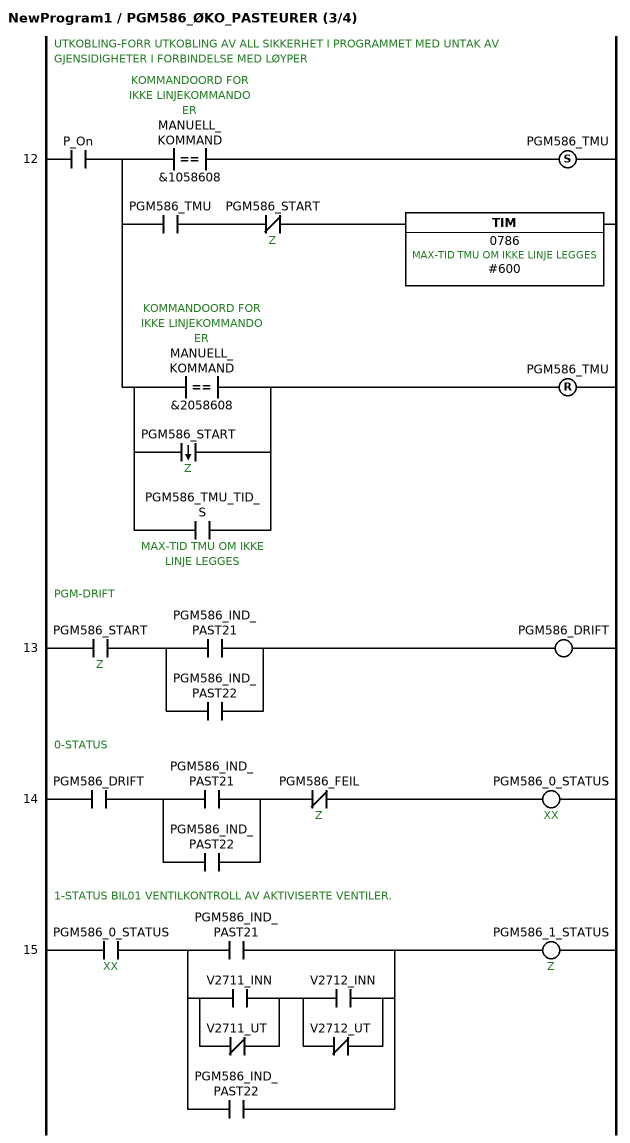
; [picture p720: NewProgram1 / PGM586_ØKO_PASTEURER, rungs 12-15]
; rung 12: UTKOBLING-FORR UTKOBLING AV ALL SIKKERHET I PROGRAMMET MED UNTAK AV GJENSIDIGHETER I FORBINDELSE MED LØYPER
LD P_On
OUT TR0
AND=L(301) MANUELL_KOMMAND &1058608  ; KOMMANDOORD FOR IKKE LINJEKOMMANDOER
SET PGM586_TMU
LD TR0
AND PGM586_TMU
ANDNOT PGM586_START  ; Z
TIM 0786 #600  ; MAX-TID TMU OM IKKE LINJE LEGGES
LD TR0
LD=L(301) MANUELL_KOMMAND &2058608  ; KOMMANDOORD FOR IKKE LINJEKOMMANDOER
%OR PGM586_START  ; Z
OR PGM586_TMU_TID_S  ; MAX-TID TMU OM IKKE LINJE LEGGES
ANDLD
RSET PGM586_TMU
; rung 13: PGM-DRIFT
LD PGM586_START  ; Z
LD PGM586_IND_PAST21
OR PGM586_IND_PAST22
ANDLD
OUT PGM586_DRIFT
; rung 14: 0-STATUS
LD PGM586_DRIFT
LD PGM586_IND_PAST21
OR PGM586_IND_PAST22
ANDLD
ANDNOT PGM586_FEIL  ; Z
OUT PGM586_0_STATUS  ; XX
; rung 15: 1-STATUS BIL01 VENTILKONTROLL AV AKTIVISERTE VENTILER.
LD PGM586_0_STATUS  ; XX
LD PGM586_IND_PAST21
LD V2711_INN
ORNOT V2711_UT
LD V2712_INN
ORNOT V2712_UT
ANDLD
ORLD
OR PGM586_IND_PAST22
ANDLD
OUT PGM586_1_STATUS  ; Z

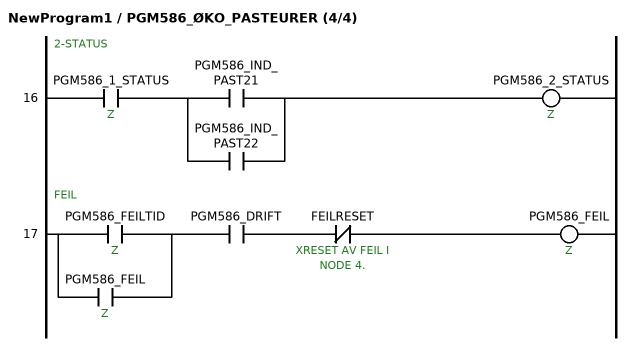
; rung 16: 2-STATUS
LD PGM586_1_STATUS  ; Z
LD PGM586_IND_PAST21
OR PGM586_IND_PAST22
ANDLD
OUT PGM586_2_STATUS  ; Z
; rung 17: FEIL
LD PGM586_FEILTID  ; Z
OR PGM586_FEIL  ; Z
AND PGM586_DRIFT
ANDNOT FEILRESET  ; XRESET AV FEIL I NODE 4.
OUT PGM586_FEIL  ; Z
; rung 18: Ingen_kommentar_funnet

### Section PGM587_RÅMELKSDRENERING

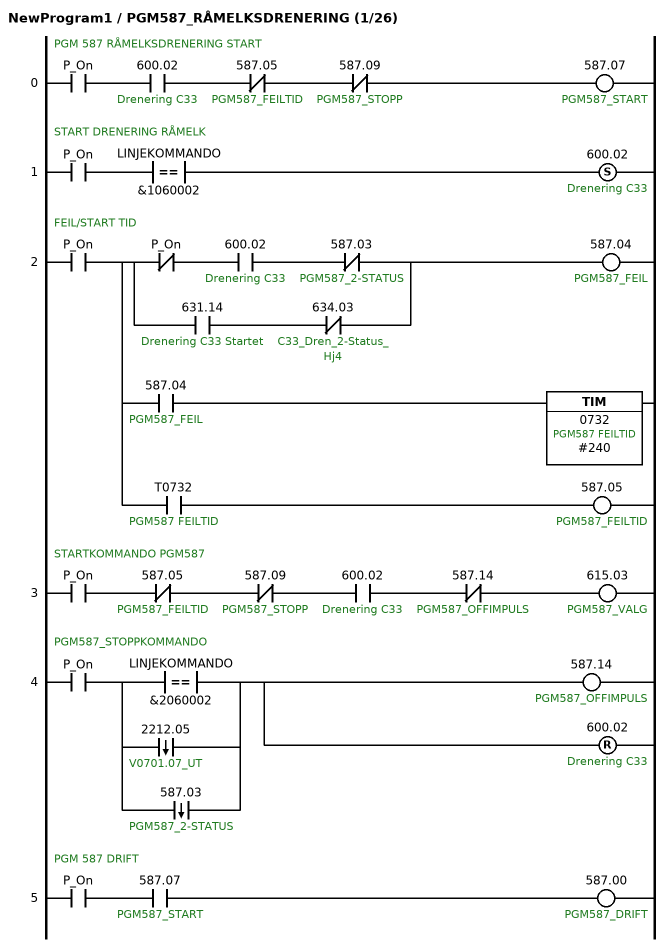
; rung 0: PGM 587 RÅMELKSDRENERING START
LD P_On
AND 600.02  ; Drenering C33
ANDNOT 587.05  ; PGM587_FEILTID
ANDNOT 587.09  ; PGM587_STOPP
OUT 587.07  ; PGM587_START
; rung 1: START DRENERING RÅMELK
LD P_On
AND=L(301) LINJEKOMMANDO &1060002
SET 600.02  ; Drenering C33
; rung 2: FEIL/START TID
LD P_On
OUT TR0
LDNOT P_On
AND 600.02  ; Drenering C33
ANDNOT 587.03  ; PGM587_2-STATUS
LD 631.14  ; Drenering C33 Startet
ANDNOT 634.03  ; C33_Dren_2-Status_Hj4
ORLD
ANDLD
OUT 587.04  ; PGM587_FEIL
LD TR0
AND 587.04  ; PGM587_FEIL
TIM 0732 #240  ; PGM587 FEILTID
LD TR0
AND T0732  ; PGM587 FEILTID
OUT 587.05  ; PGM587_FEILTID
; rung 3: STARTKOMMANDO PGM587
LD P_On
ANDNOT 587.05  ; PGM587_FEILTID
ANDNOT 587.09  ; PGM587_STOPP
AND 600.02  ; Drenering C33
ANDNOT 587.14  ; PGM587_OFFIMPULS
OUT 615.03  ; PGM587_VALG
; rung 4: PGM587_STOPPKOMMANDO
LD P_On
LD=L(301) LINJEKOMMANDO &2060002
%OR 2212.05  ; V0701.07_UT
%OR 587.03  ; PGM587_2-STATUS
ANDLD
OUT 587.14  ; PGM587_OFFIMPULS
RSET 600.02  ; Drenering C33
; rung 5: PGM 587 DRIFT
LD P_On
AND 587.07  ; PGM587_START
OUT 587.00  ; PGM587_DRIFT

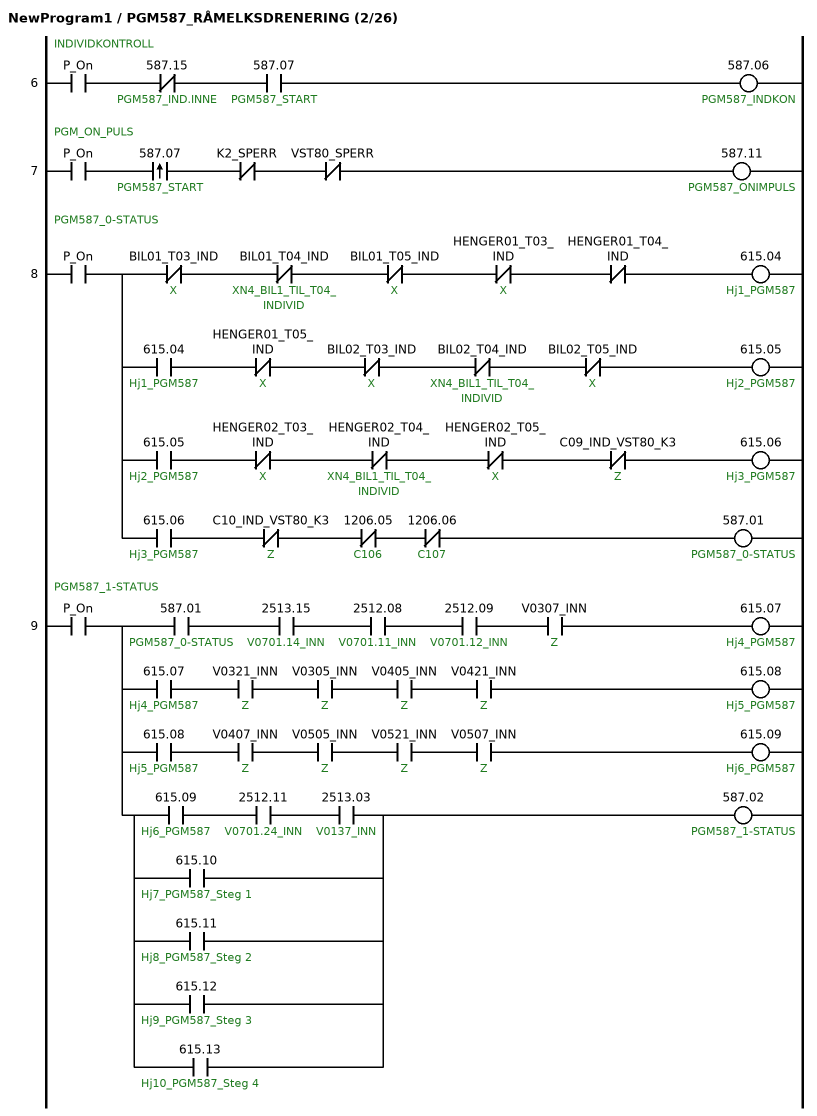
; rung 6: INDIVIDKONTROLL
LD P_On
ANDNOT 587.15  ; PGM587_IND.INNE
AND 587.07  ; PGM587_START
OUT 587.06  ; PGM587_INDKON
; rung 7: PGM_ON_PULS
LD P_On
@AND 587.07  ; PGM587_START
ANDNOT K2_SPERR
ANDNOT VST80_SPERR
OUT 587.11  ; PGM587_ONIMPULS
; rung 8: PGM587_0-STATUS
LD P_On
OUT TR0
ANDNOT BIL01_T03_IND  ; X
ANDNOT BIL01_T04_IND  ; XN4_BIL1_TIL_T04_INDIVID
ANDNOT BIL01_T05_IND  ; X
ANDNOT HENGER01_T03_IND  ; X
ANDNOT HENGER01_T04_IND
OUT 615.04  ; Hj1_PGM587
LD TR0
AND 615.04  ; Hj1_PGM587
ANDNOT HENGER01_T05_IND  ; X
ANDNOT BIL02_T03_IND  ; X
ANDNOT BIL02_T04_IND  ; XN4_BIL1_TIL_T04_INDIVID
ANDNOT BIL02_T05_IND  ; X
OUT 615.05  ; Hj2_PGM587
LD TR0
AND 615.05  ; Hj2_PGM587
ANDNOT HENGER02_T03_IND  ; X
ANDNOT HENGER02_T04_IND  ; XN4_BIL1_TIL_T04_INDIVID
ANDNOT HENGER02_T05_IND  ; X
ANDNOT C09_IND_VST80_K3  ; Z
OUT 615.06  ; Hj3_PGM587
LD TR0
AND 615.06  ; Hj3_PGM587
ANDNOT C10_IND_VST80_K3  ; Z
ANDNOT 1206.05  ; C106
ANDNOT 1206.06  ; C107
OUT 587.01  ; PGM587_0-STATUS
; rung 9: PGM587_1-STATUS
LD P_On
OUT TR0
AND 587.01  ; PGM587_0-STATUS
AND 2513.15  ; V0701.14_INN
AND 2512.08  ; V0701.11_INN
AND 2512.09  ; V0701.12_INN
AND V0307_INN  ; Z
OUT 615.07  ; Hj4_PGM587
LD TR0
AND 615.07  ; Hj4_PGM587
AND V0321_INN  ; Z
AND V0305_INN  ; Z
AND V0405_INN  ; Z
AND V0421_INN  ; Z
OUT 615.08  ; Hj5_PGM587
LD TR0
AND 615.08  ; Hj5_PGM587
AND V0407_INN  ; Z
AND V0505_INN  ; Z
AND V0521_INN  ; Z
AND V0507_INN  ; Z
OUT 615.09  ; Hj6_PGM587
LD TR0
LD 615.09  ; Hj6_PGM587
AND 2512.11  ; V0701.24_INN
AND 2513.03  ; V0137_INN
OR 615.10  ; Hj7_PGM587_Steg 1
OR 615.11  ; Hj8_PGM587_Steg 2
OR 615.12  ; Hj9_PGM587_Steg 3
OR 615.13  ; Hj10_PGM587_Steg 4
ANDLD
OUT 587.02  ; PGM587_1-STATUS

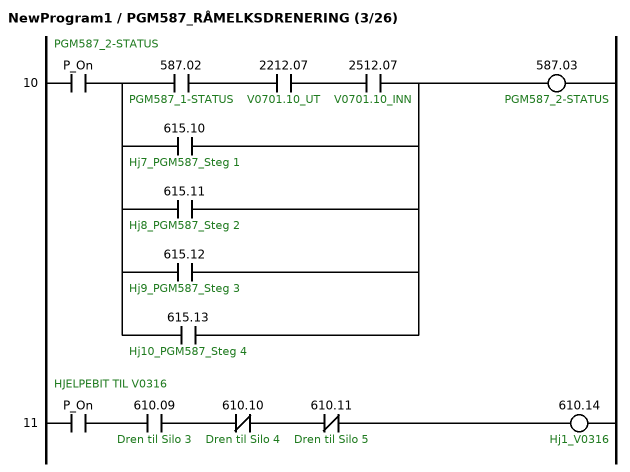
; rung 10: PGM587_2-STATUS
LD P_On
LD 587.02  ; PGM587_1-STATUS
AND 2212.07  ; V0701.10_UT
AND 2512.07  ; V0701.10_INN
OR 615.10  ; Hj7_PGM587_Steg 1
OR 615.11  ; Hj8_PGM587_Steg 2
OR 615.12  ; Hj9_PGM587_Steg 3
OR 615.13  ; Hj10_PGM587_Steg 4
ANDLD
OUT 587.03  ; PGM587_2-STATUS
; rung 11: HJELPEBIT TIL V0316
LD P_On
AND 610.09  ; Dren til Silo 3
ANDNOT 610.10  ; Dren til Silo 4
ANDNOT 610.11  ; Dren til Silo 5
OUT 610.14  ; Hj1_V0316

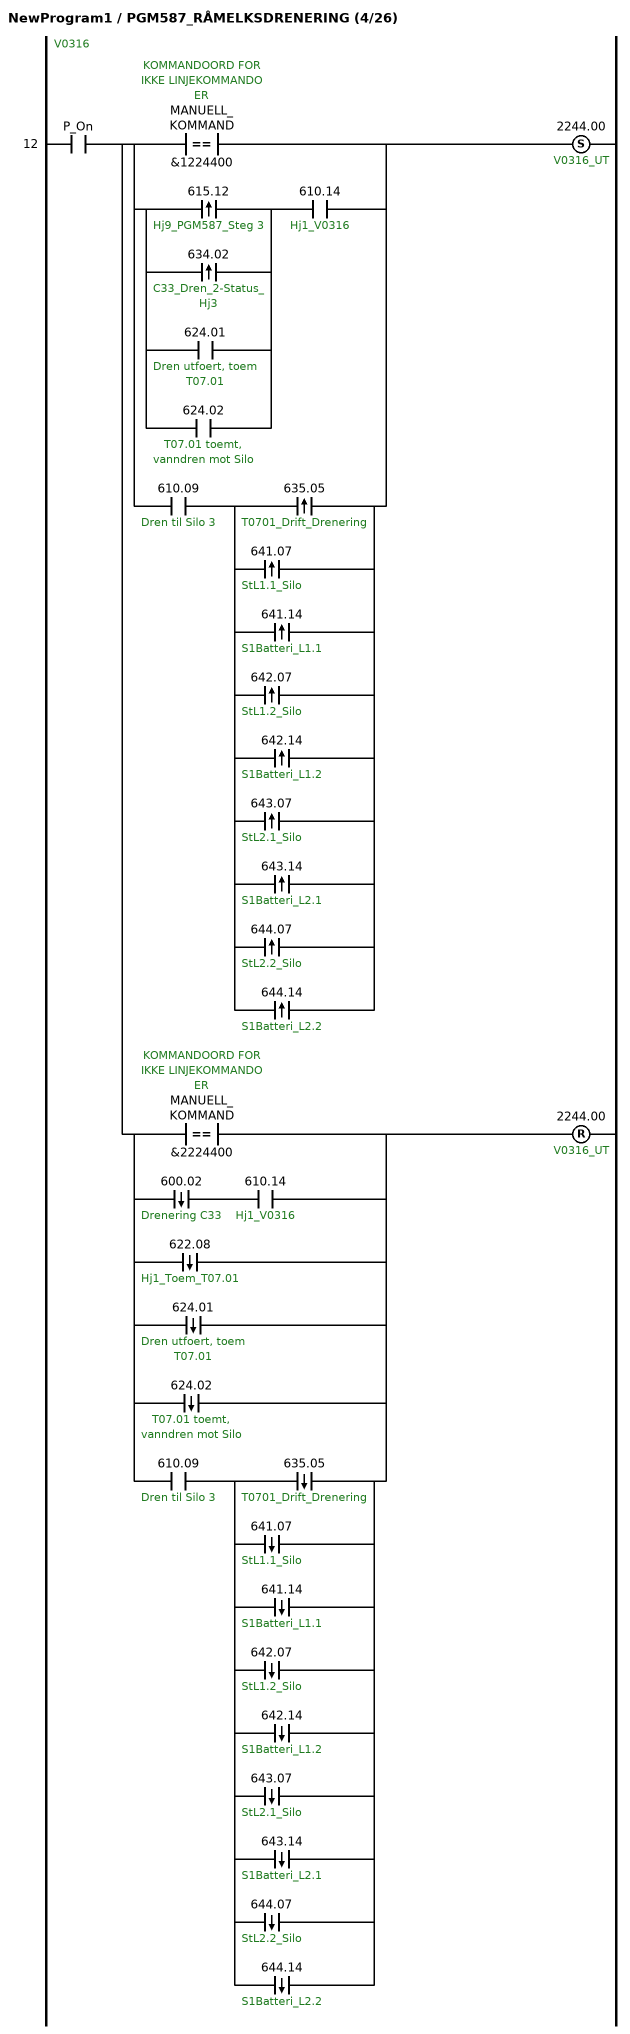
; rung 12: V0316
LD P_On
OUT TR0
LD=L(301) MANUELL_KOMMAND &1224400  ; KOMMANDOORD FOR IKKE LINJEKOMMANDOER
@LD 615.12  ; Hj9_PGM587_Steg 3
@OR 634.02  ; C33_Dren_2-Status_Hj3
OR 624.01  ; Dren utfoert, toem T07.01
OR 624.02  ; T07.01 toemt, vanndren mot Silo
AND 610.14  ; Hj1_V0316
ORLD
LD 610.09  ; Dren til Silo 3
@LD 635.05  ; T0701_Drift_Drenering
@OR 641.07  ; StL1.1_Silo
@OR 641.14  ; S1Batteri_L1.1
@OR 642.07  ; StL1.2_Silo
@OR 642.14  ; S1Batteri_L1.2
@OR 643.07  ; StL2.1_Silo
@OR 643.14  ; S1Batteri_L2.1
@OR 644.07  ; StL2.2_Silo
@OR 644.14  ; S1Batteri_L2.2
ANDLD
ORLD
ANDLD
SET 2244.00  ; V0316_UT
LD TR0
LD=L(301) MANUELL_KOMMAND &2224400  ; KOMMANDOORD FOR IKKE LINJEKOMMANDOER
%LD 600.02  ; Drenering C33
AND 610.14  ; Hj1_V0316
ORLD
%OR 622.08  ; Hj1_Toem_T07.01
%OR 624.01  ; Dren utfoert, toem T07.01
%OR 624.02  ; T07.01 toemt, vanndren mot Silo
LD 610.09  ; Dren til Silo 3
%LD 635.05  ; T0701_Drift_Drenering
%OR 641.07  ; StL1.1_Silo
%OR 641.14  ; S1Batteri_L1.1
%OR 642.07  ; StL1.2_Silo
%OR 642.14  ; S1Batteri_L1.2
%OR 643.07  ; StL2.1_Silo
%OR 643.14  ; S1Batteri_L2.1
%OR 644.07  ; StL2.2_Silo
%OR 644.14  ; S1Batteri_L2.2
ANDLD
ORLD
ANDLD
RSET 2244.00  ; V0316_UT

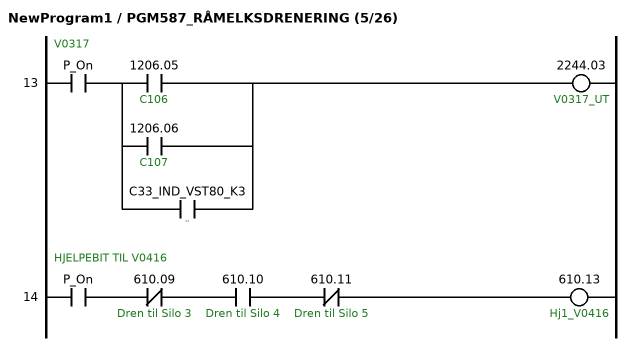
; rung 13: V0317
LD P_On
LD 1206.05  ; C106
OR 1206.06  ; C107
OR C33_IND_VST80_K3  ; ¨
ANDLD
OUT 2244.03  ; V0317_UT
; rung 14: HJELPEBIT TIL V0416
LD P_On
ANDNOT 610.09  ; Dren til Silo 3
AND 610.10  ; Dren til Silo 4
ANDNOT 610.11  ; Dren til Silo 5
OUT 610.13  ; Hj1_V0416

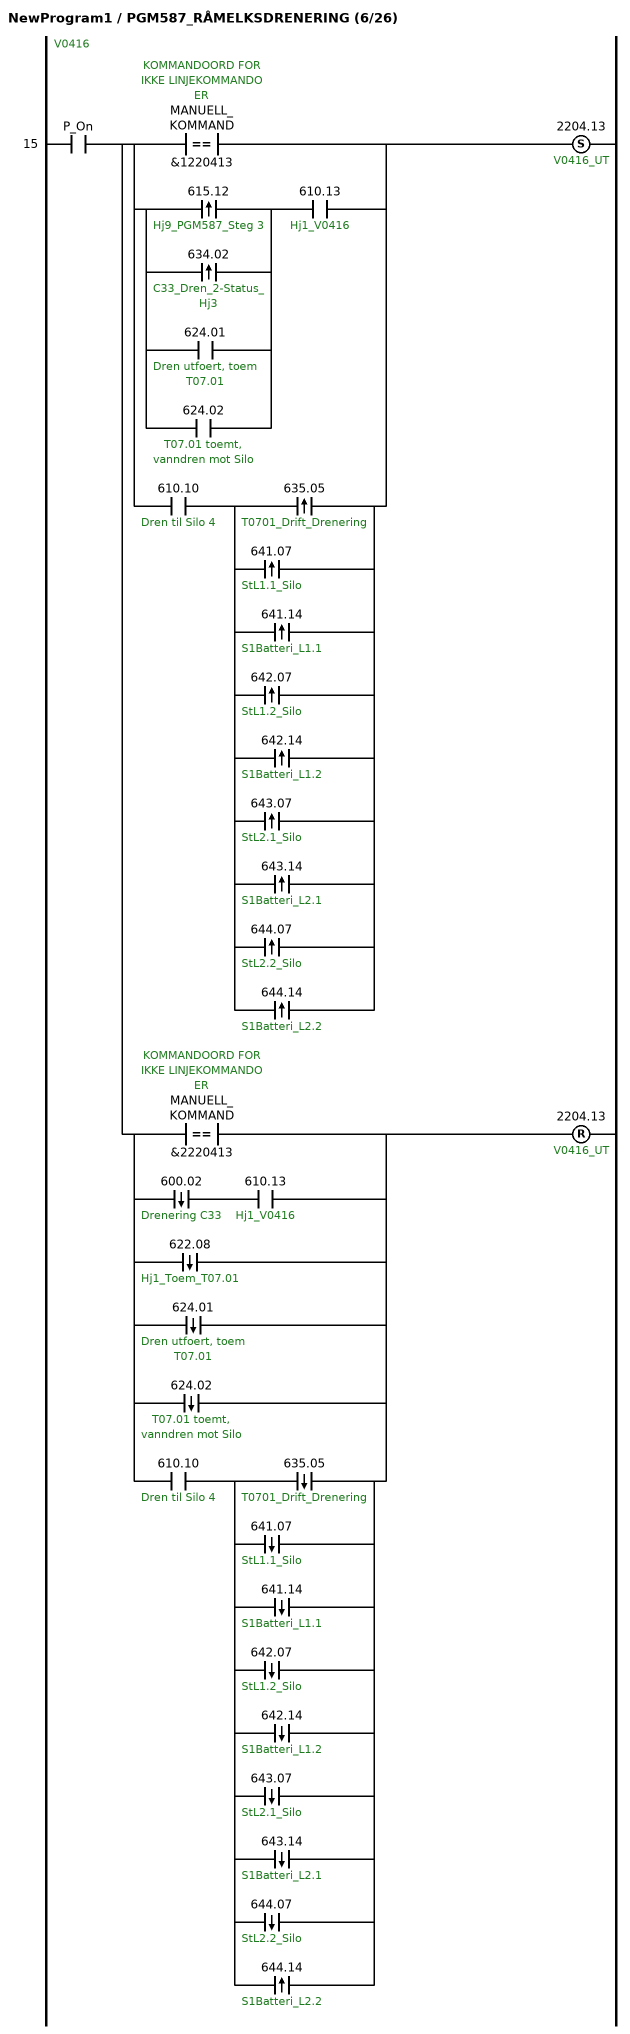
; rung 15: V0416
LD P_On
OUT TR0
LD=L(301) MANUELL_KOMMAND &1220413  ; KOMMANDOORD FOR IKKE LINJEKOMMANDOER
@LD 615.12  ; Hj9_PGM587_Steg 3
@OR 634.02  ; C33_Dren_2-Status_Hj3
OR 624.01  ; Dren utfoert, toem T07.01
OR 624.02  ; T07.01 toemt, vanndren mot Silo
AND 610.13  ; Hj1_V0416
ORLD
LD 610.10  ; Dren til Silo 4
@LD 635.05  ; T0701_Drift_Drenering
@OR 641.07  ; StL1.1_Silo
@OR 641.14  ; S1Batteri_L1.1
@OR 642.07  ; StL1.2_Silo
@OR 642.14  ; S1Batteri_L1.2
@OR 643.07  ; StL2.1_Silo
@OR 643.14  ; S1Batteri_L2.1
@OR 644.07  ; StL2.2_Silo
@OR 644.14  ; S1Batteri_L2.2
ANDLD
ORLD
ANDLD
SET 2204.13  ; V0416_UT
LD TR0
LD=L(301) MANUELL_KOMMAND &2220413  ; KOMMANDOORD FOR IKKE LINJEKOMMANDOER
%LD 600.02  ; Drenering C33
AND 610.13  ; Hj1_V0416
ORLD
%OR 622.08  ; Hj1_Toem_T07.01
%OR 624.01  ; Dren utfoert, toem T07.01
%OR 624.02  ; T07.01 toemt, vanndren mot Silo
LD 610.10  ; Dren til Silo 4
%LD 635.05  ; T0701_Drift_Drenering
%OR 641.07  ; StL1.1_Silo
%OR 641.14  ; S1Batteri_L1.1
%OR 642.07  ; StL1.2_Silo
%OR 642.14  ; S1Batteri_L1.2
%OR 643.07  ; StL2.1_Silo
%OR 643.14  ; S1Batteri_L2.1
%OR 644.07  ; StL2.2_Silo
@OR 644.14  ; S1Batteri_L2.2
ANDLD
ORLD
ANDLD
RSET 2204.13  ; V0416_UT

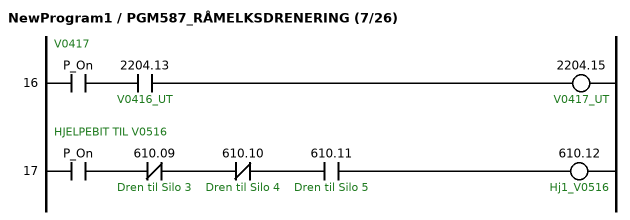
; rung 16: V0417
LD P_On
AND 2204.13  ; V0416_UT
OUT 2204.15  ; V0417_UT
; rung 17: HJELPEBIT TIL V0516
LD P_On
ANDNOT 610.09  ; Dren til Silo 3
ANDNOT 610.10  ; Dren til Silo 4
AND 610.11  ; Dren til Silo 5
OUT 610.12  ; Hj1_V0516

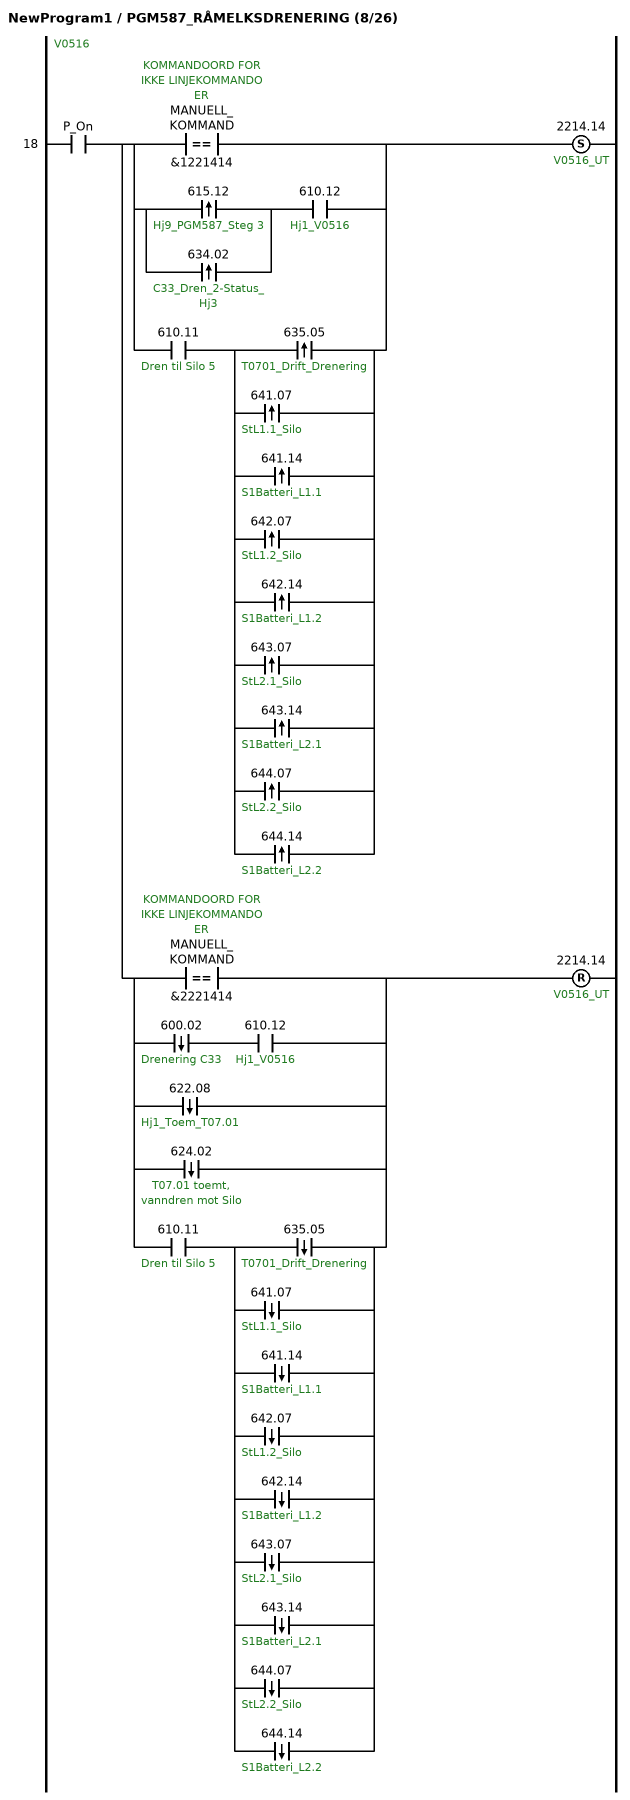
; rung 18: V0516
LD P_On
OUT TR0
LD=L(301) MANUELL_KOMMAND &1221414  ; KOMMANDOORD FOR IKKE LINJEKOMMANDOER
@LD 615.12  ; Hj9_PGM587_Steg 3
@OR 634.02  ; C33_Dren_2-Status_Hj3
AND 610.12  ; Hj1_V0516
ORLD
LD 610.11  ; Dren til Silo 5
@LD 635.05  ; T0701_Drift_Drenering
@OR 641.07  ; StL1.1_Silo
@OR 641.14  ; S1Batteri_L1.1
@OR 642.07  ; StL1.2_Silo
@OR 642.14  ; S1Batteri_L1.2
@OR 643.07  ; StL2.1_Silo
@OR 643.14  ; S1Batteri_L2.1
@OR 644.07  ; StL2.2_Silo
@OR 644.14  ; S1Batteri_L2.2
ANDLD
ORLD
ANDLD
SET 2214.14  ; V0516_UT
LD TR0
LD=L(301) MANUELL_KOMMAND &2221414  ; KOMMANDOORD FOR IKKE LINJEKOMMANDOER
%LD 600.02  ; Drenering C33
AND 610.12  ; Hj1_V0516
ORLD
%OR 622.08  ; Hj1_Toem_T07.01
%OR 624.02  ; T07.01 toemt, vanndren mot Silo
LD 610.11  ; Dren til Silo 5
%LD 635.05  ; T0701_Drift_Drenering
%OR 641.07  ; StL1.1_Silo
%OR 641.14  ; S1Batteri_L1.1
%OR 642.07  ; StL1.2_Silo
%OR 642.14  ; S1Batteri_L1.2
%OR 643.07  ; StL2.1_Silo
%OR 643.14  ; S1Batteri_L2.1
%OR 644.07  ; StL2.2_Silo
%OR 644.14  ; S1Batteri_L2.2
ANDLD
ORLD
ANDLD
RSET 2214.14  ; V0516_UT

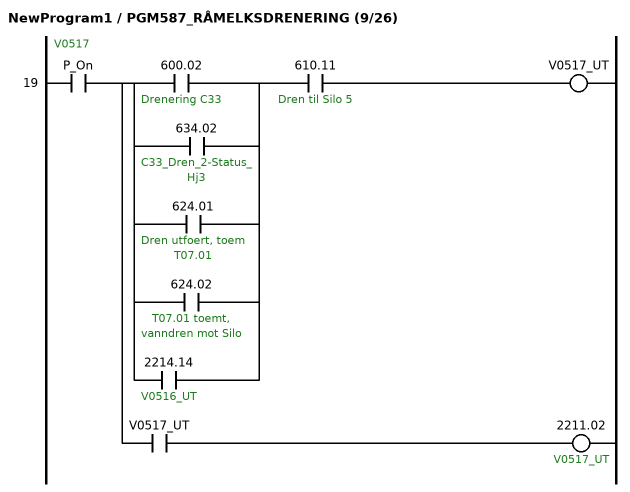
; rung 19: V0517
LD P_On
OUT TR0
LD 600.02  ; Drenering C33
OR 634.02  ; C33_Dren_2-Status_Hj3
OR 624.01  ; Dren utfoert, toem T07.01
OR 624.02  ; T07.01 toemt, vanndren mot Silo
OR 2214.14  ; V0516_UT
ANDLD
AND 610.11  ; Dren til Silo 5
OUT V0517_UT
LD TR0
AND V0517_UT
OUT 2211.02  ; V0517_UT

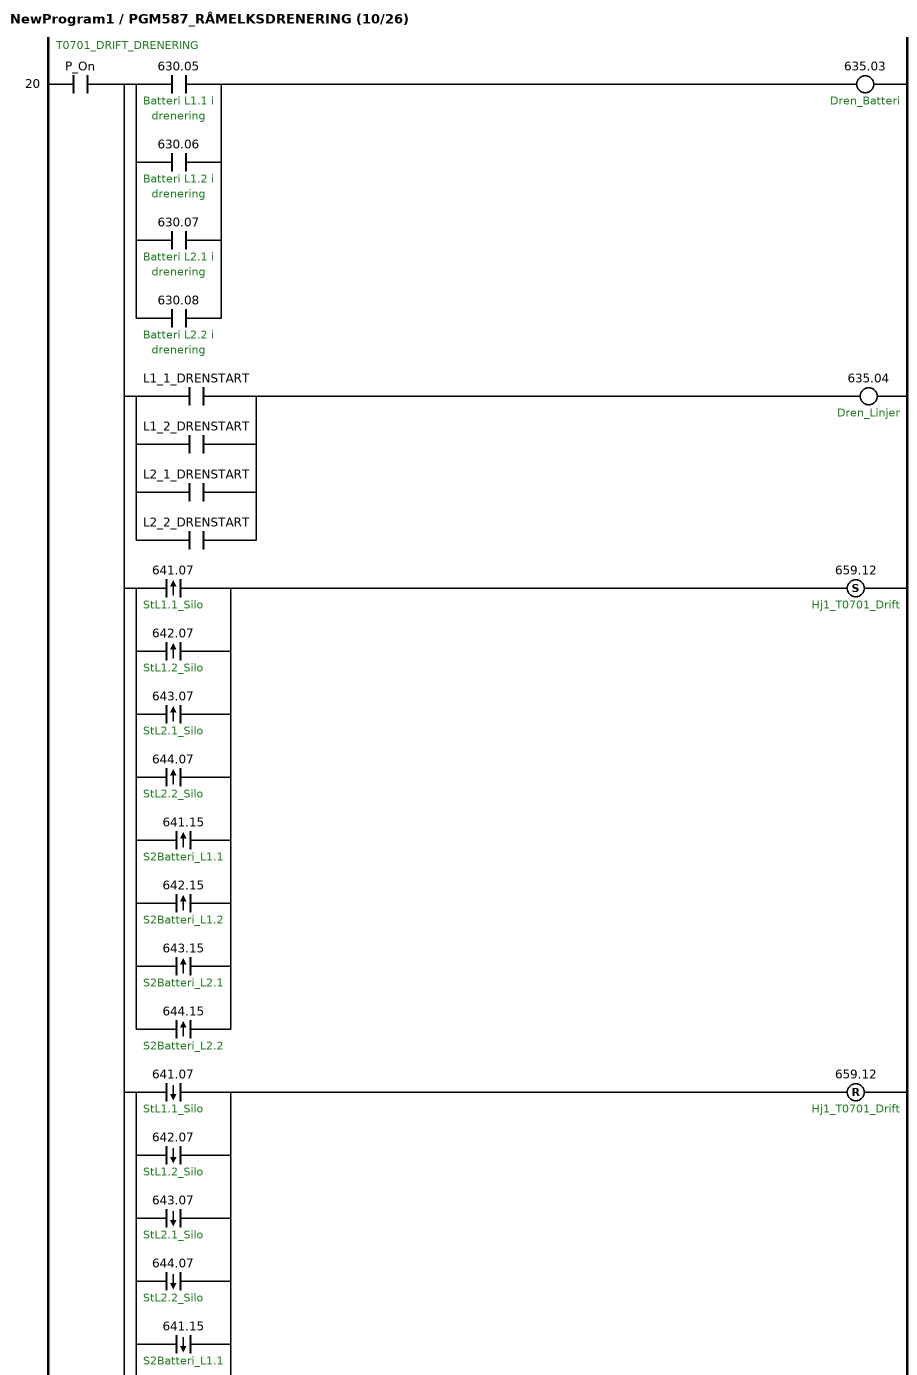

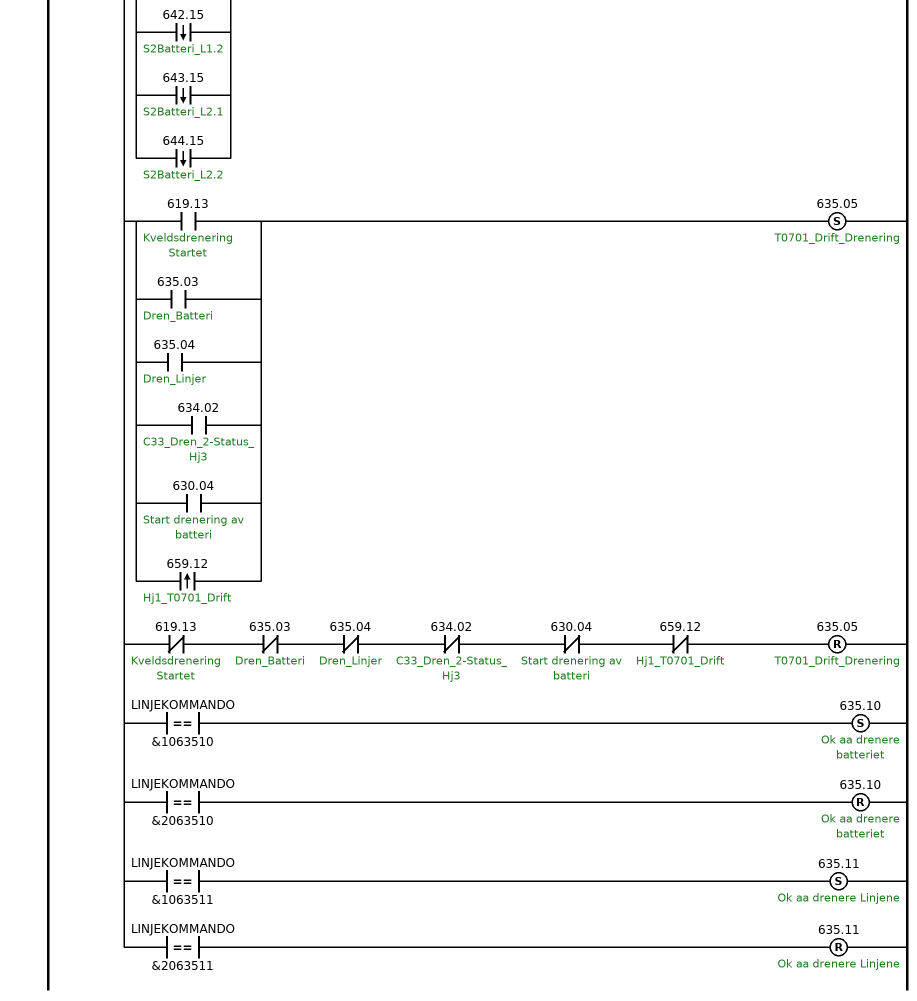
; rung 20: T0701_DRIFT_DRENERING
LD P_On
OUT TR0
LD 630.05  ; Batteri L1.1 i drenering
OR 630.06  ; Batteri L1.2 i drenering
OR 630.07  ; Batteri L2.1 i drenering
OR 630.08  ; Batteri L2.2 i drenering
ANDLD
OUT 635.03  ; Dren_Batteri
LD TR0
LD L1_1_DRENSTART
OR L1_2_DRENSTART
OR L2_1_DRENSTART
OR L2_2_DRENSTART
ANDLD
OUT 635.04  ; Dren_Linjer
LD TR0
@LD 641.07  ; StL1.1_Silo
@OR 642.07  ; StL1.2_Silo
@OR 643.07  ; StL2.1_Silo
@OR 644.07  ; StL2.2_Silo
@OR 641.15  ; S2Batteri_L1.1
@OR 642.15  ; S2Batteri_L1.2
@OR 643.15  ; S2Batteri_L2.1
@OR 644.15  ; S2Batteri_L2.2
ANDLD
SET 659.12  ; Hj1_T0701_Drift
LD TR0
%LD 641.07  ; StL1.1_Silo
%OR 642.07  ; StL1.2_Silo
%OR 643.07  ; StL2.1_Silo
%OR 644.07  ; StL2.2_Silo
%OR 641.15  ; S2Batteri_L1.1
%OR 642.15  ; S2Batteri_L1.2
%OR 643.15  ; S2Batteri_L2.1
%OR 644.15  ; S2Batteri_L2.2
ANDLD
RSET 659.12  ; Hj1_T0701_Drift
LD TR0
LD 619.13  ; Kveldsdrenering Startet
OR 635.03  ; Dren_Batteri
OR 635.04  ; Dren_Linjer
OR 634.02  ; C33_Dren_2-Status_Hj3
OR 630.04  ; Start drenering av batteri
@OR 659.12  ; Hj1_T0701_Drift
ANDLD
SET 635.05  ; T0701_Drift_Drenering
LD TR0
ANDNOT 619.13  ; Kveldsdrenering Startet
ANDNOT 635.03  ; Dren_Batteri
ANDNOT 635.04  ; Dren_Linjer
ANDNOT 634.02  ; C33_Dren_2-Status_Hj3
ANDNOT 630.04  ; Start drenering av batteri
ANDNOT 659.12  ; Hj1_T0701_Drift
RSET 635.05  ; T0701_Drift_Drenering
LD TR0
AND=L(301) LINJEKOMMANDO &1063510
SET 635.10  ; Ok aa drenere batteriet
LD TR0
AND=L(301) LINJEKOMMANDO &2063510
RSET 635.10  ; Ok aa drenere batteriet
LD TR0
AND=L(301) LINJEKOMMANDO &1063511
SET 635.11  ; Ok aa drenere Linjene
LD TR0
AND=L(301) LINJEKOMMANDO &2063511
RSET 635.11  ; Ok aa drenere Linjene

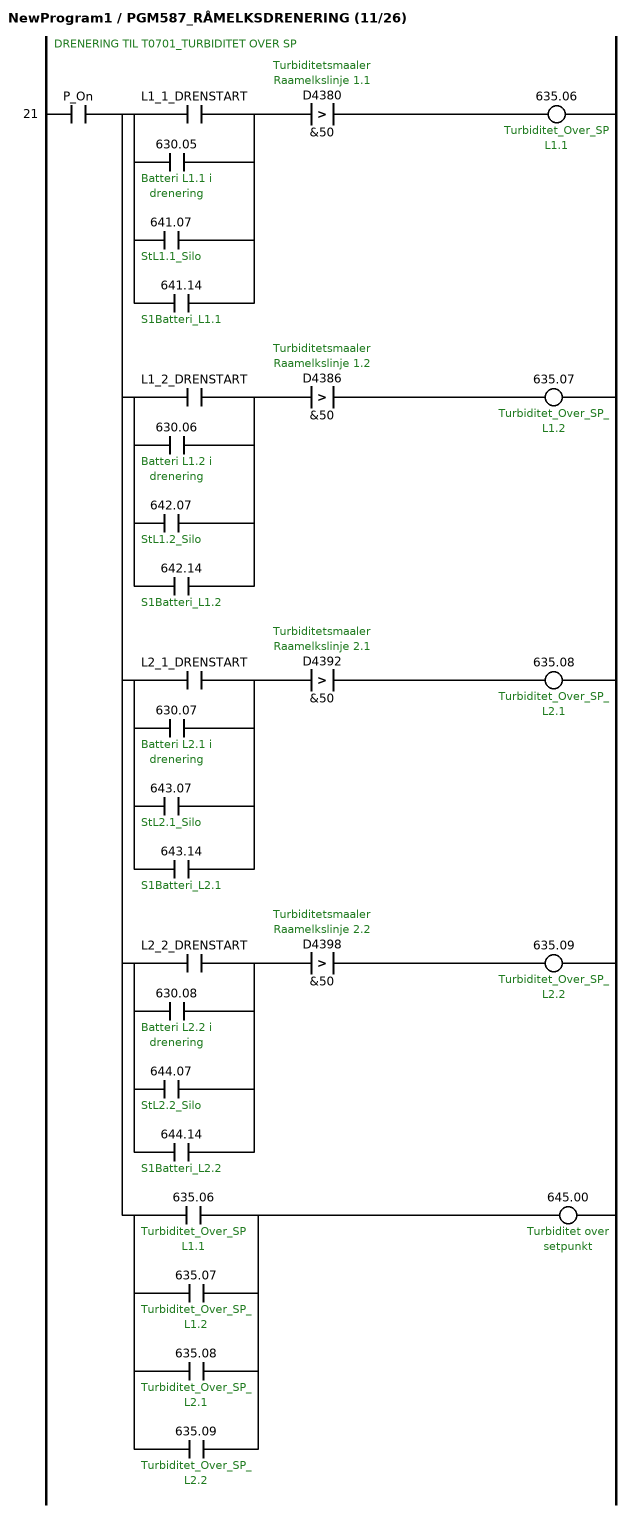
; rung 21: DRENERING TIL T0701_TURBIDITET OVER SP
LD P_On
OUT TR0
LD L1_1_DRENSTART
OR 630.05  ; Batteri L1.1 i drenering
OR 641.07  ; StL1.1_Silo
OR 641.14  ; S1Batteri_L1.1
ANDLD
AND>(320) D4380 &50  ; Turbiditetsmaaler Raamelkslinje 1.1
OUT 635.06  ; Turbiditet_Over_SP L1.1
LD TR0
LD L1_2_DRENSTART
OR 630.06  ; Batteri L1.2 i drenering
OR 642.07  ; StL1.2_Silo
OR 642.14  ; S1Batteri_L1.2
ANDLD
AND>(320) D4386 &50  ; Turbiditetsmaaler Raamelkslinje 1.2
OUT 635.07  ; Turbiditet_Over_SP_L1.2
LD TR0
LD L2_1_DRENSTART
OR 630.07  ; Batteri L2.1 i drenering
OR 643.07  ; StL2.1_Silo
OR 643.14  ; S1Batteri_L2.1
ANDLD
AND>(320) D4392 &50  ; Turbiditetsmaaler Raamelkslinje 2.1
OUT 635.08  ; Turbiditet_Over_SP_L2.1
LD TR0
LD L2_2_DRENSTART
OR 630.08  ; Batteri L2.2 i drenering
OR 644.07  ; StL2.2_Silo
OR 644.14  ; S1Batteri_L2.2
ANDLD
AND>(320) D4398 &50  ; Turbiditetsmaaler Raamelkslinje 2.2
OUT 635.09  ; Turbiditet_Over_SP_L2.2
LD TR0
LD 635.06  ; Turbiditet_Over_SP L1.1
OR 635.07  ; Turbiditet_Over_SP_L1.2
OR 635.08  ; Turbiditet_Over_SP_L2.1
OR 635.09  ; Turbiditet_Over_SP_L2.2
ANDLD
OUT 645.00  ; Turbiditet over setpunkt

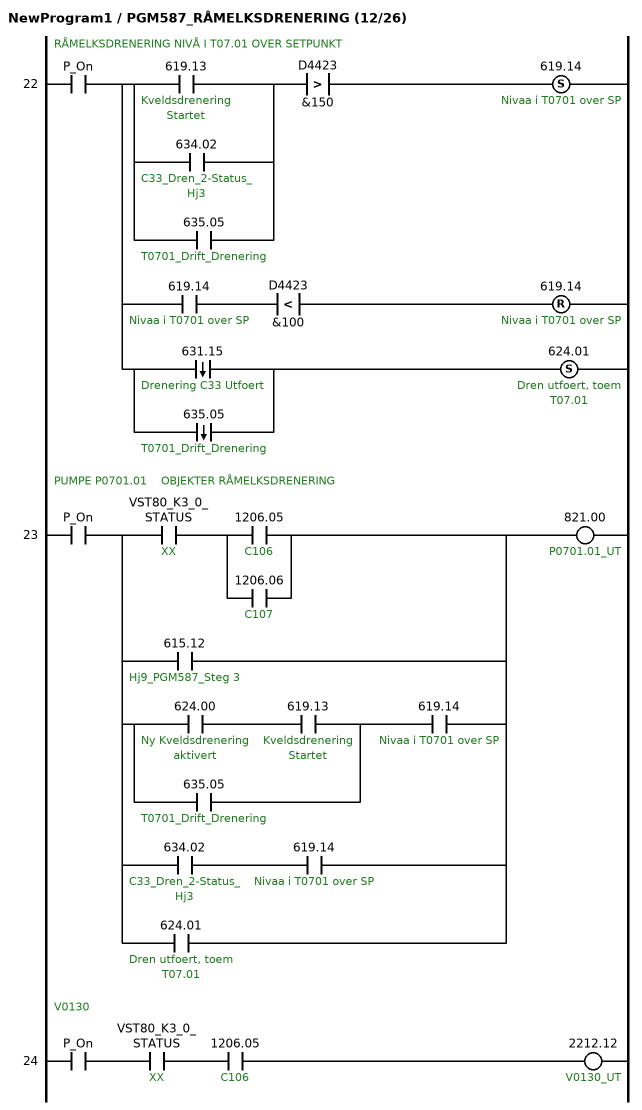
; rung 22: RÅMELKSDRENERING NIVÅ I T07.01 OVER SETPUNKT
LD P_On
OUT TR0
LD 619.13  ; Kveldsdrenering Startet
OR 634.02  ; C33_Dren_2-Status_Hj3
OR 635.05  ; T0701_Drift_Drenering
ANDLD
AND>(320) D4423 &150
SET 619.14  ; Nivaa i T0701 over SP
LD TR0
AND 619.14  ; Nivaa i T0701 over SP
AND<(310) D4423 &100
RSET 619.14  ; Nivaa i T0701 over SP
LD TR0
%LD 631.15  ; Drenering C33 Utfoert
%OR 635.05  ; T0701_Drift_Drenering
ANDLD
SET 624.01  ; Dren utfoert, toem T07.01
; rung 23: PUMPE P0701.01    OBJEKTER RÅMELKSDRENERING
LD P_On
LD VST80_K3_0_STATUS  ; XX
LD 1206.05  ; C106
OR 1206.06  ; C107
ANDLD
OR 615.12  ; Hj9_PGM587_Steg 3
LD 624.00  ; Ny Kveldsdrenering aktivert
AND 619.13  ; Kveldsdrenering Startet
OR 635.05  ; T0701_Drift_Drenering
AND 619.14  ; Nivaa i T0701 over SP
ORLD
LD 634.02  ; C33_Dren_2-Status_Hj3
AND 619.14  ; Nivaa i T0701 over SP
ORLD
OR 624.01  ; Dren utfoert, toem T07.01
ANDLD
OUT 821.00  ; P0701.01_UT
; rung 24: V0130
LD P_On
AND VST80_K3_0_STATUS  ; XX
AND 1206.05  ; C106
OUT 2212.12  ; V0130_UT

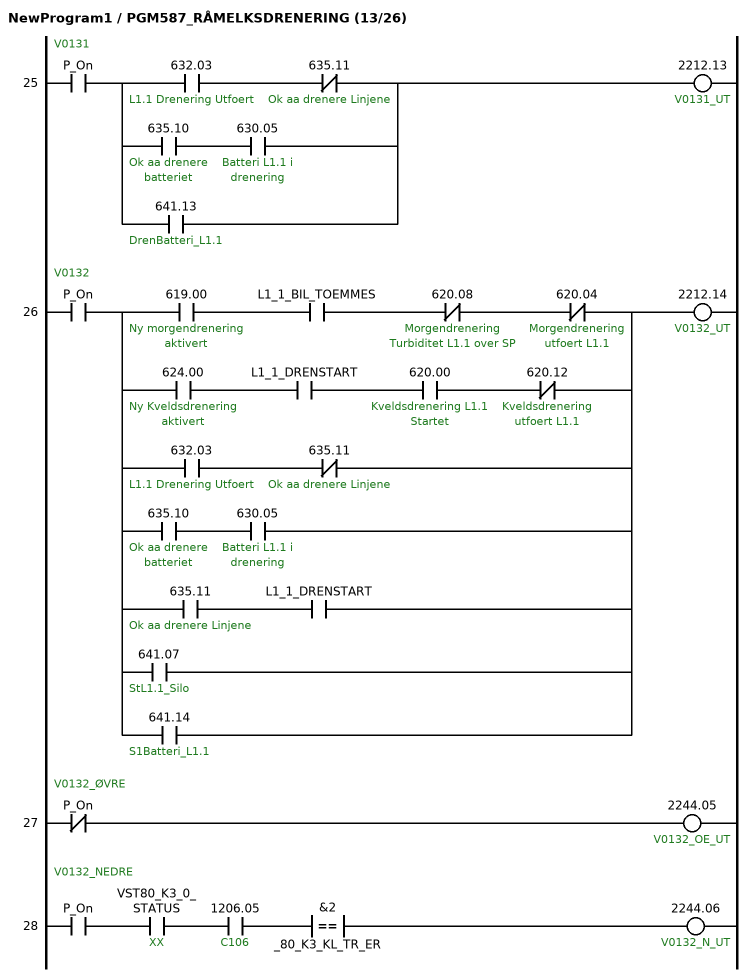
; rung 25: V0131
LD P_On
LD 632.03  ; L1.1 Drenering Utfoert
ANDNOT 635.11  ; Ok aa drenere Linjene
LD 635.10  ; Ok aa drenere batteriet
AND 630.05  ; Batteri L1.1 i drenering
ORLD
OR 641.13  ; DrenBatteri_L1.1
ANDLD
OUT 2212.13  ; V0131_UT
; rung 26: V0132
LD P_On
LD 619.00  ; Ny morgendrenering aktivert
AND L1_1_BIL_TOEMMES
ANDNOT 620.08  ; Morgendrenering Turbiditet L1.1 over SP
ANDNOT 620.04  ; Morgendrenering utfoert L1.1
LD 624.00  ; Ny Kveldsdrenering aktivert
AND L1_1_DRENSTART
AND 620.00  ; Kveldsdrenering L1.1 Startet
ANDNOT 620.12  ; Kveldsdrenering utfoert L1.1
ORLD
LD 632.03  ; L1.1 Drenering Utfoert
ANDNOT 635.11  ; Ok aa drenere Linjene
ORLD
LD 635.10  ; Ok aa drenere batteriet
AND 630.05  ; Batteri L1.1 i drenering
ORLD
LD 635.11  ; Ok aa drenere Linjene
AND L1_1_DRENSTART
ORLD
OR 641.07  ; StL1.1_Silo
OR 641.14  ; S1Batteri_L1.1
ANDLD
OUT 2212.14  ; V0132_UT
; rung 27: V0132_ØVRE
LDNOT P_On
OUT 2244.05  ; V0132_OE_UT
; rung 28: V0132_NEDRE
LD P_On
AND VST80_K3_0_STATUS  ; XX
AND 1206.05  ; C106
AND=(300) &2 _80_K3_KL_TR_ER
OUT 2244.06  ; V0132_N_UT

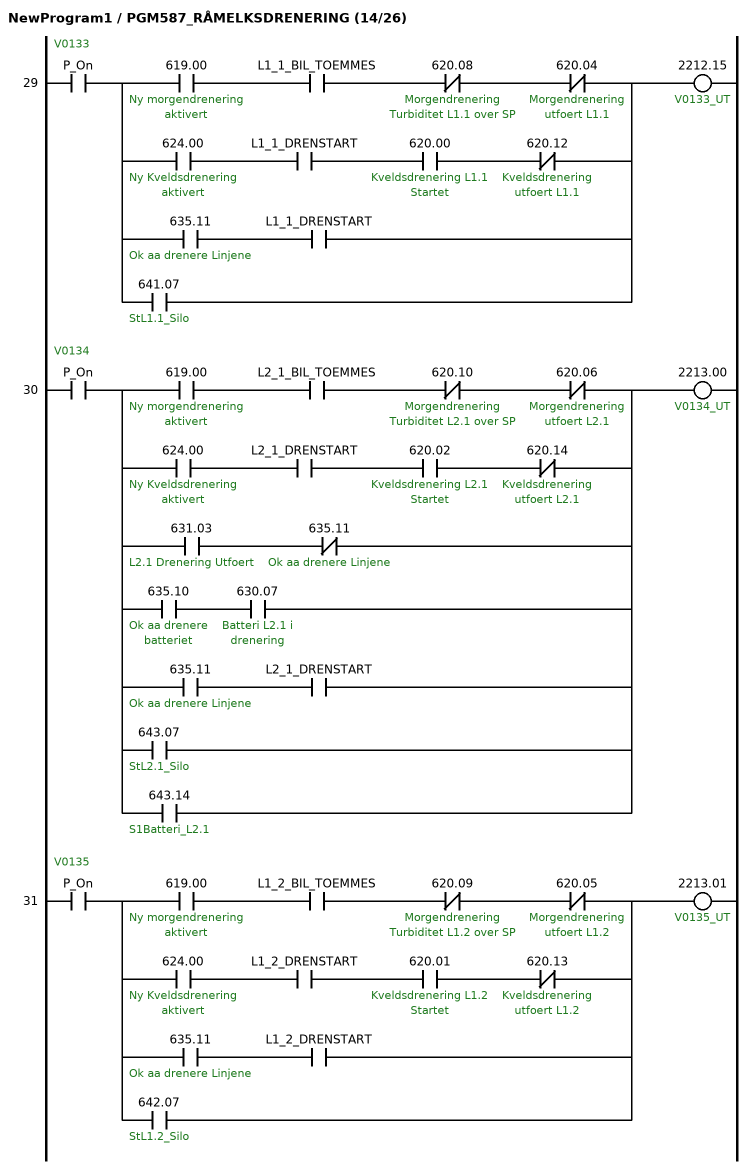
; rung 29: V0133
LD P_On
LD 619.00  ; Ny morgendrenering aktivert
AND L1_1_BIL_TOEMMES
ANDNOT 620.08  ; Morgendrenering Turbiditet L1.1 over SP
ANDNOT 620.04  ; Morgendrenering utfoert L1.1
LD 624.00  ; Ny Kveldsdrenering aktivert
AND L1_1_DRENSTART
AND 620.00  ; Kveldsdrenering L1.1 Startet
ANDNOT 620.12  ; Kveldsdrenering utfoert L1.1
ORLD
LD 635.11  ; Ok aa drenere Linjene
AND L1_1_DRENSTART
ORLD
OR 641.07  ; StL1.1_Silo
ANDLD
OUT 2212.15  ; V0133_UT
; rung 30: V0134
LD P_On
LD 619.00  ; Ny morgendrenering aktivert
AND L2_1_BIL_TOEMMES
ANDNOT 620.10  ; Morgendrenering Turbiditet L2.1 over SP
ANDNOT 620.06  ; Morgendrenering utfoert L2.1
LD 624.00  ; Ny Kveldsdrenering aktivert
AND L2_1_DRENSTART
AND 620.02  ; Kveldsdrenering L2.1 Startet
ANDNOT 620.14  ; Kveldsdrenering utfoert L2.1
ORLD
LD 631.03  ; L2.1 Drenering Utfoert
ANDNOT 635.11  ; Ok aa drenere Linjene
ORLD
LD 635.10  ; Ok aa drenere batteriet
AND 630.07  ; Batteri L2.1 i drenering
ORLD
LD 635.11  ; Ok aa drenere Linjene
AND L2_1_DRENSTART
ORLD
OR 643.07  ; StL2.1_Silo
OR 643.14  ; S1Batteri_L2.1
ANDLD
OUT 2213.00  ; V0134_UT
; rung 31: V0135
LD P_On
LD 619.00  ; Ny morgendrenering aktivert
AND L1_2_BIL_TOEMMES
ANDNOT 620.09  ; Morgendrenering Turbiditet L1.2 over SP
ANDNOT 620.05  ; Morgendrenering utfoert L1.2
LD 624.00  ; Ny Kveldsdrenering aktivert
AND L1_2_DRENSTART
AND 620.01  ; Kveldsdrenering L1.2 Startet
ANDNOT 620.13  ; Kveldsdrenering utfoert L1.2
ORLD
LD 635.11  ; Ok aa drenere Linjene
AND L1_2_DRENSTART
ORLD
OR 642.07  ; StL1.2_Silo
ANDLD
OUT 2213.01  ; V0135_UT

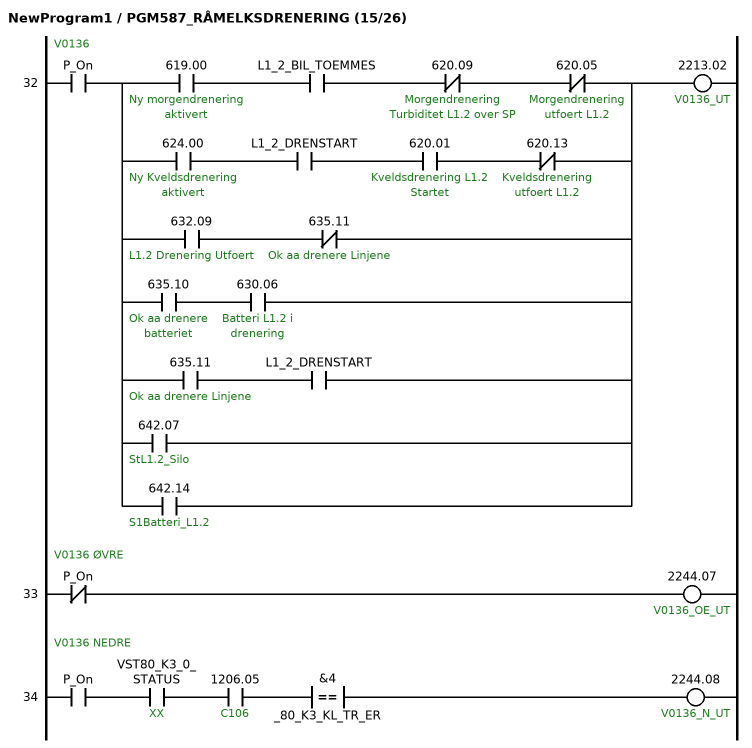
; rung 32: V0136
LD P_On
LD 619.00  ; Ny morgendrenering aktivert
AND L1_2_BIL_TOEMMES
ANDNOT 620.09  ; Morgendrenering Turbiditet L1.2 over SP
ANDNOT 620.05  ; Morgendrenering utfoert L1.2
LD 624.00  ; Ny Kveldsdrenering aktivert
AND L1_2_DRENSTART
AND 620.01  ; Kveldsdrenering L1.2 Startet
ANDNOT 620.13  ; Kveldsdrenering utfoert L1.2
ORLD
LD 632.09  ; L1.2 Drenering Utfoert
ANDNOT 635.11  ; Ok aa drenere Linjene
ORLD
LD 635.10  ; Ok aa drenere batteriet
AND 630.06  ; Batteri L1.2 i drenering
ORLD
LD 635.11  ; Ok aa drenere Linjene
AND L1_2_DRENSTART
ORLD
OR 642.07  ; StL1.2_Silo
OR 642.14  ; S1Batteri_L1.2
ANDLD
OUT 2213.02  ; V0136_UT
; rung 33: V0136 ØVRE
LDNOT P_On
OUT 2244.07  ; V0136_OE_UT
; rung 34: V0136 NEDRE
LD P_On
AND VST80_K3_0_STATUS  ; XX
AND 1206.05  ; C106
AND=(300) &4 _80_K3_KL_TR_ER
OUT 2244.08  ; V0136_N_UT

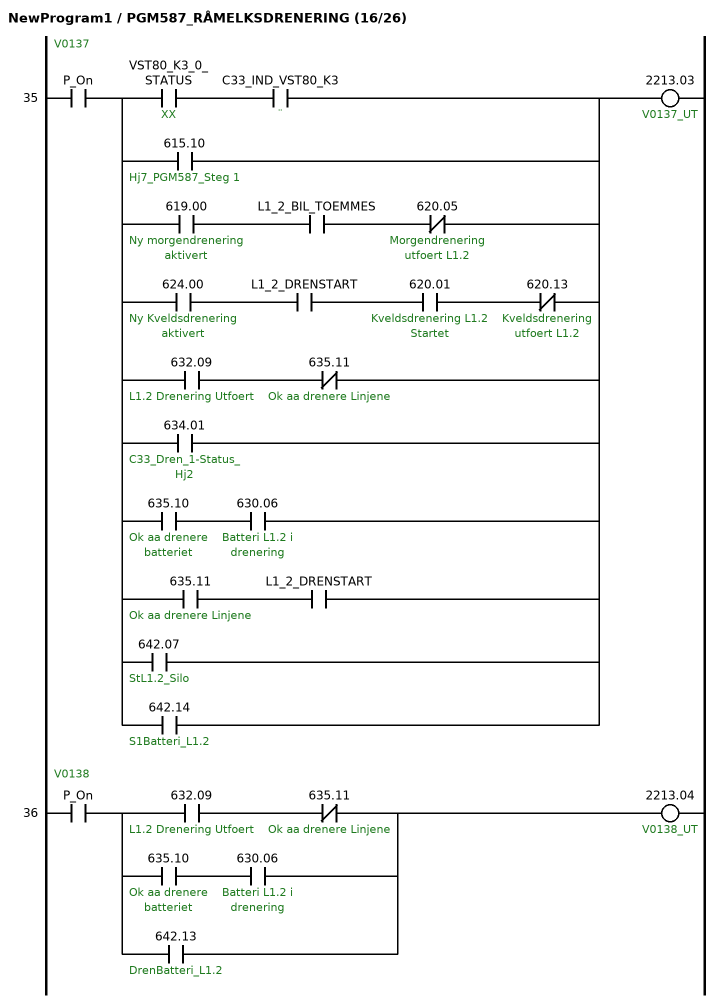
; rung 35: V0137
LD P_On
LD VST80_K3_0_STATUS  ; XX
AND C33_IND_VST80_K3  ; ¨
OR 615.10  ; Hj7_PGM587_Steg 1
LD 619.00  ; Ny morgendrenering aktivert
AND L1_2_BIL_TOEMMES
ANDNOT 620.05  ; Morgendrenering utfoert L1.2
ORLD
LD 624.00  ; Ny Kveldsdrenering aktivert
AND L1_2_DRENSTART
AND 620.01  ; Kveldsdrenering L1.2 Startet
ANDNOT 620.13  ; Kveldsdrenering utfoert L1.2
ORLD
LD 632.09  ; L1.2 Drenering Utfoert
ANDNOT 635.11  ; Ok aa drenere Linjene
ORLD
OR 634.01  ; C33_Dren_1-Status_Hj2
LD 635.10  ; Ok aa drenere batteriet
AND 630.06  ; Batteri L1.2 i drenering
ORLD
LD 635.11  ; Ok aa drenere Linjene
AND L1_2_DRENSTART
ORLD
OR 642.07  ; StL1.2_Silo
OR 642.14  ; S1Batteri_L1.2
ANDLD
OUT 2213.03  ; V0137_UT
; rung 36: V0138
LD P_On
LD 632.09  ; L1.2 Drenering Utfoert
ANDNOT 635.11  ; Ok aa drenere Linjene
LD 635.10  ; Ok aa drenere batteriet
AND 630.06  ; Batteri L1.2 i drenering
ORLD
OR 642.13  ; DrenBatteri_L1.2
ANDLD
OUT 2213.04  ; V0138_UT

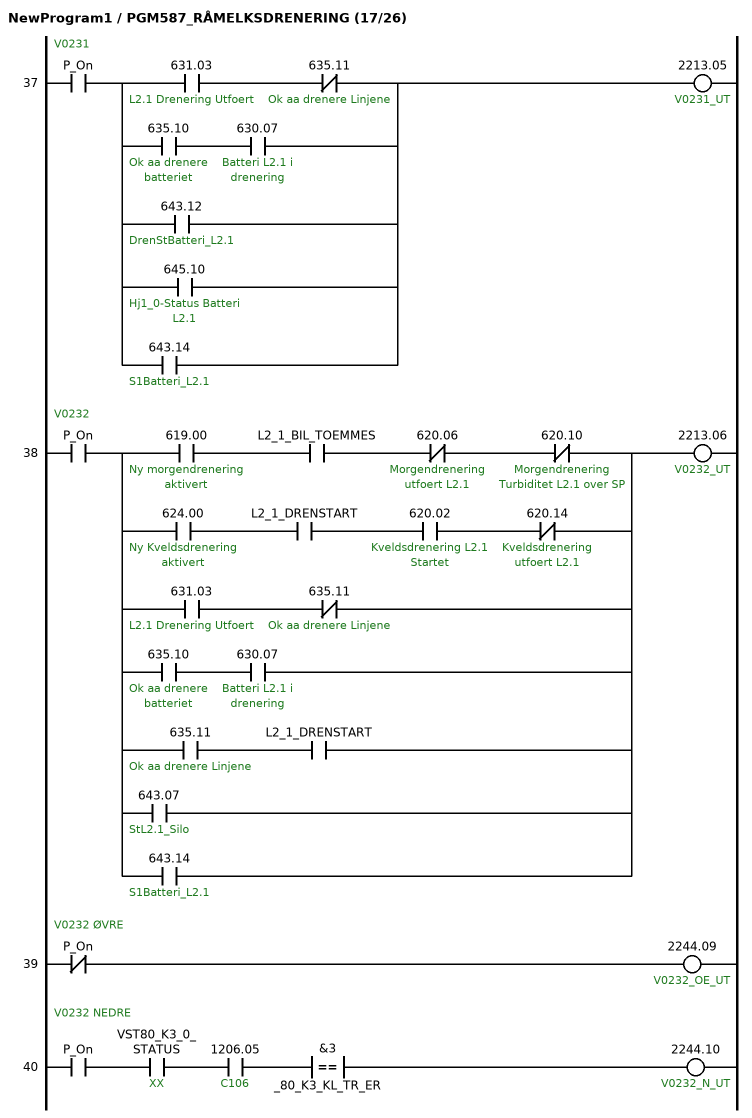
; rung 37: V0231
LD P_On
LD 631.03  ; L2.1 Drenering Utfoert
ANDNOT 635.11  ; Ok aa drenere Linjene
LD 635.10  ; Ok aa drenere batteriet
AND 630.07  ; Batteri L2.1 i drenering
ORLD
OR 643.12  ; DrenStBatteri_L2.1
OR 645.10  ; Hj1_0-Status Batteri L2.1
OR 643.14  ; S1Batteri_L2.1
ANDLD
OUT 2213.05  ; V0231_UT
; rung 38: V0232
LD P_On
LD 619.00  ; Ny morgendrenering aktivert
AND L2_1_BIL_TOEMMES
ANDNOT 620.06  ; Morgendrenering utfoert L2.1
ANDNOT 620.10  ; Morgendrenering Turbiditet L2.1 over SP
LD 624.00  ; Ny Kveldsdrenering aktivert
AND L2_1_DRENSTART
AND 620.02  ; Kveldsdrenering L2.1 Startet
ANDNOT 620.14  ; Kveldsdrenering utfoert L2.1
ORLD
LD 631.03  ; L2.1 Drenering Utfoert
ANDNOT 635.11  ; Ok aa drenere Linjene
ORLD
LD 635.10  ; Ok aa drenere batteriet
AND 630.07  ; Batteri L2.1 i drenering
ORLD
LD 635.11  ; Ok aa drenere Linjene
AND L2_1_DRENSTART
ORLD
OR 643.07  ; StL2.1_Silo
OR 643.14  ; S1Batteri_L2.1
ANDLD
OUT 2213.06  ; V0232_UT
; rung 39: V0232 ØVRE
LDNOT P_On
OUT 2244.09  ; V0232_OE_UT
; rung 40: V0232 NEDRE
LD P_On
AND VST80_K3_0_STATUS  ; XX
AND 1206.05  ; C106
AND=(300) &3 _80_K3_KL_TR_ER
OUT 2244.10  ; V0232_N_UT

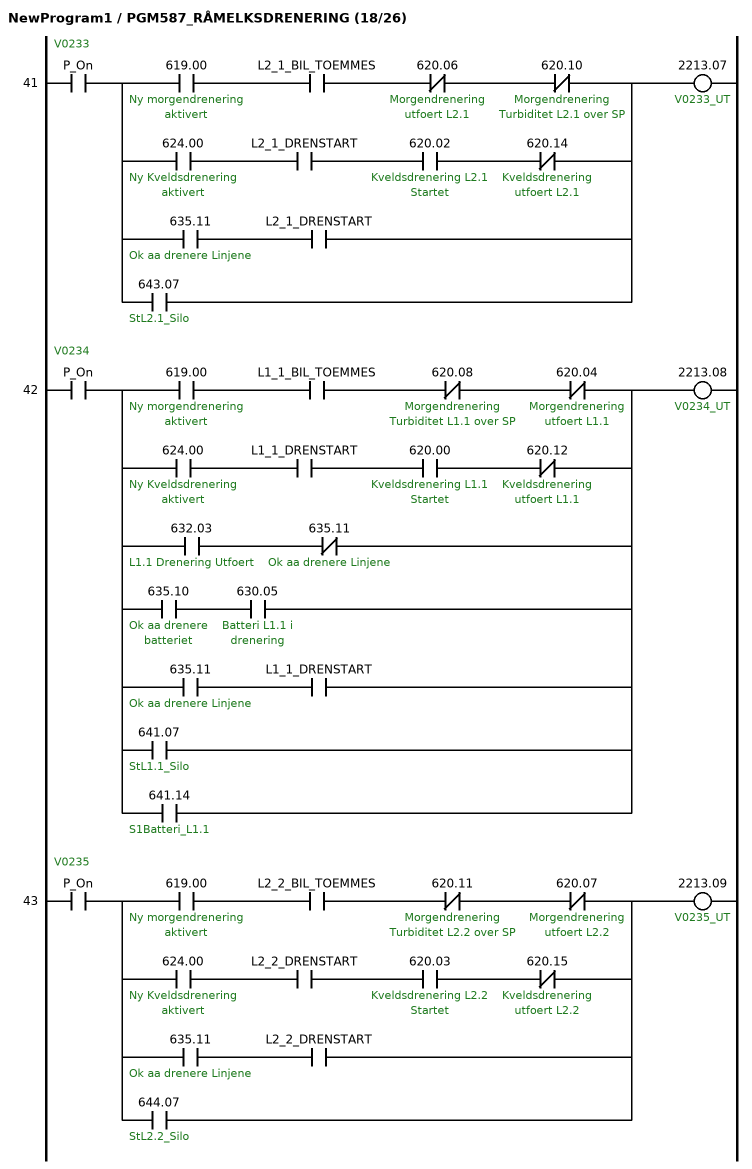
; rung 41: V0233
LD P_On
LD 619.00  ; Ny morgendrenering aktivert
AND L2_1_BIL_TOEMMES
ANDNOT 620.06  ; Morgendrenering utfoert L2.1
ANDNOT 620.10  ; Morgendrenering Turbiditet L2.1 over SP
LD 624.00  ; Ny Kveldsdrenering aktivert
AND L2_1_DRENSTART
AND 620.02  ; Kveldsdrenering L2.1 Startet
ANDNOT 620.14  ; Kveldsdrenering utfoert L2.1
ORLD
LD 635.11  ; Ok aa drenere Linjene
AND L2_1_DRENSTART
ORLD
OR 643.07  ; StL2.1_Silo
ANDLD
OUT 2213.07  ; V0233_UT
; rung 42: V0234
LD P_On
LD 619.00  ; Ny morgendrenering aktivert
AND L1_1_BIL_TOEMMES
ANDNOT 620.08  ; Morgendrenering Turbiditet L1.1 over SP
ANDNOT 620.04  ; Morgendrenering utfoert L1.1
LD 624.00  ; Ny Kveldsdrenering aktivert
AND L1_1_DRENSTART
AND 620.00  ; Kveldsdrenering L1.1 Startet
ANDNOT 620.12  ; Kveldsdrenering utfoert L1.1
ORLD
LD 632.03  ; L1.1 Drenering Utfoert
ANDNOT 635.11  ; Ok aa drenere Linjene
ORLD
LD 635.10  ; Ok aa drenere batteriet
AND 630.05  ; Batteri L1.1 i drenering
ORLD
LD 635.11  ; Ok aa drenere Linjene
AND L1_1_DRENSTART
ORLD
OR 641.07  ; StL1.1_Silo
OR 641.14  ; S1Batteri_L1.1
ANDLD
OUT 2213.08  ; V0234_UT
; rung 43: V0235
LD P_On
LD 619.00  ; Ny morgendrenering aktivert
AND L2_2_BIL_TOEMMES
ANDNOT 620.11  ; Morgendrenering Turbiditet L2.2 over SP
ANDNOT 620.07  ; Morgendrenering utfoert L2.2
LD 624.00  ; Ny Kveldsdrenering aktivert
AND L2_2_DRENSTART
AND 620.03  ; Kveldsdrenering L2.2 Startet
ANDNOT 620.15  ; Kveldsdrenering utfoert L2.2
ORLD
LD 635.11  ; Ok aa drenere Linjene
AND L2_2_DRENSTART
ORLD
OR 644.07  ; StL2.2_Silo
ANDLD
OUT 2213.09  ; V0235_UT

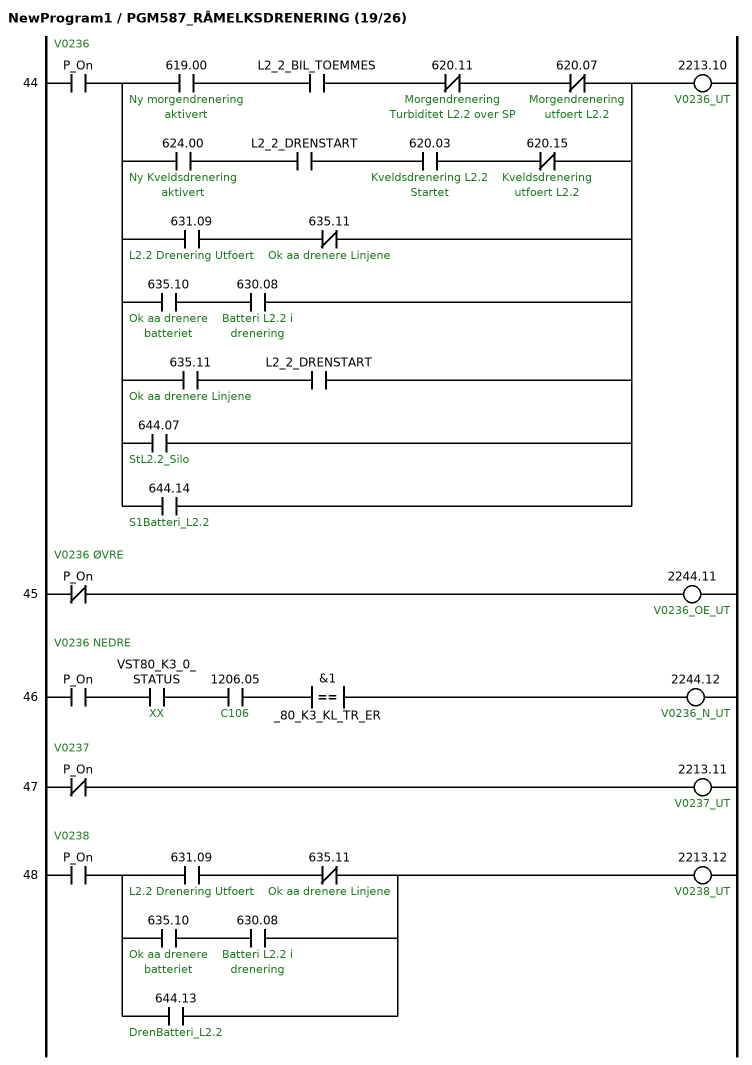
; rung 44: V0236
LD P_On
LD 619.00  ; Ny morgendrenering aktivert
AND L2_2_BIL_TOEMMES
ANDNOT 620.11  ; Morgendrenering Turbiditet L2.2 over SP
ANDNOT 620.07  ; Morgendrenering utfoert L2.2
LD 624.00  ; Ny Kveldsdrenering aktivert
AND L2_2_DRENSTART
AND 620.03  ; Kveldsdrenering L2.2 Startet
ANDNOT 620.15  ; Kveldsdrenering utfoert L2.2
ORLD
LD 631.09  ; L2.2 Drenering Utfoert
ANDNOT 635.11  ; Ok aa drenere Linjene
ORLD
LD 635.10  ; Ok aa drenere batteriet
AND 630.08  ; Batteri L2.2 i drenering
ORLD
LD 635.11  ; Ok aa drenere Linjene
AND L2_2_DRENSTART
ORLD
OR 644.07  ; StL2.2_Silo
OR 644.14  ; S1Batteri_L2.2
ANDLD
OUT 2213.10  ; V0236_UT
; rung 45: V0236 ØVRE
LDNOT P_On
OUT 2244.11  ; V0236_OE_UT
; rung 46: V0236 NEDRE
LD P_On
AND VST80_K3_0_STATUS  ; XX
AND 1206.05  ; C106
AND=(300) &1 _80_K3_KL_TR_ER
OUT 2244.12  ; V0236_N_UT
; rung 47: V0237
LDNOT P_On
OUT 2213.11  ; V0237_UT
; rung 48: V0238
LD P_On
LD 631.09  ; L2.2 Drenering Utfoert
ANDNOT 635.11  ; Ok aa drenere Linjene
LD 635.10  ; Ok aa drenere batteriet
AND 630.08  ; Batteri L2.2 i drenering
ORLD
OR 644.13  ; DrenBatteri_L2.2
ANDLD
OUT 2213.12  ; V0238_UT

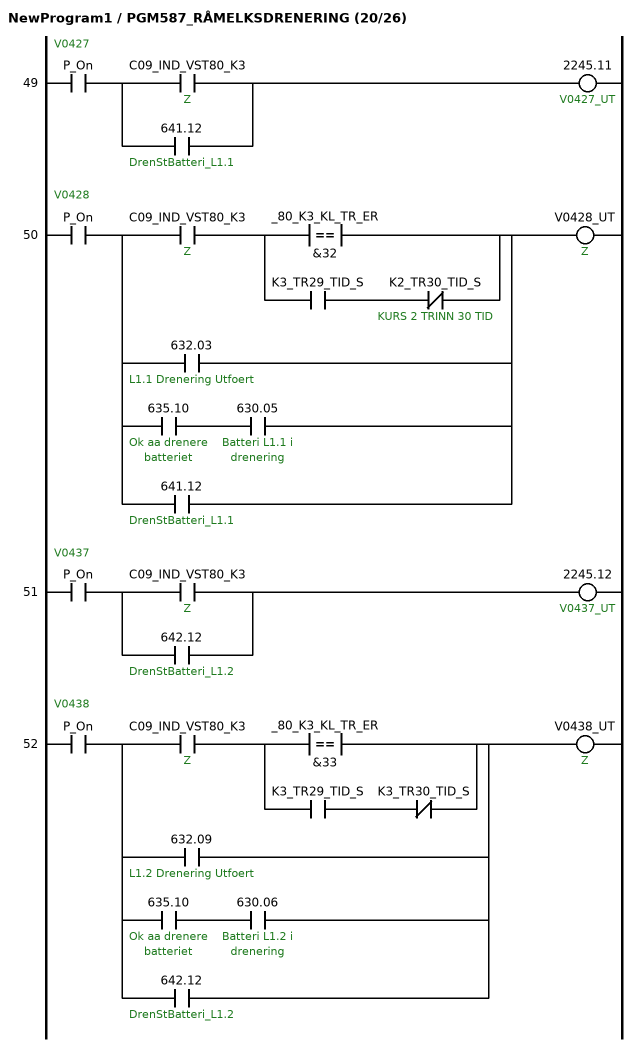
; rung 49: V0427
LD P_On
LD C09_IND_VST80_K3  ; Z
OR 641.12  ; DrenStBatteri_L1.1
ANDLD
OUT 2245.11  ; V0427_UT
; rung 50: V0428
LD P_On
LD C09_IND_VST80_K3  ; Z
LD=(300) _80_K3_KL_TR_ER &32
LD K3_TR29_TID_S
ANDNOT K2_TR30_TID_S  ; KURS 2 TRINN 30 TID
ORLD
ANDLD
OR 632.03  ; L1.1 Drenering Utfoert
LD 635.10  ; Ok aa drenere batteriet
AND 630.05  ; Batteri L1.1 i drenering
ORLD
OR 641.12  ; DrenStBatteri_L1.1
ANDLD
OUT V0428_UT  ; Z
; rung 51: V0437
LD P_On
LD C09_IND_VST80_K3  ; Z
OR 642.12  ; DrenStBatteri_L1.2
ANDLD
OUT 2245.12  ; V0437_UT
; rung 52: V0438
LD P_On
LD C09_IND_VST80_K3  ; Z
LD=(300) _80_K3_KL_TR_ER &33
LD K3_TR29_TID_S
ANDNOT K3_TR30_TID_S
ORLD
ANDLD
OR 632.09  ; L1.2 Drenering Utfoert
LD 635.10  ; Ok aa drenere batteriet
AND 630.06  ; Batteri L1.2 i drenering
ORLD
OR 642.12  ; DrenStBatteri_L1.2
ANDLD
OUT V0438_UT  ; Z

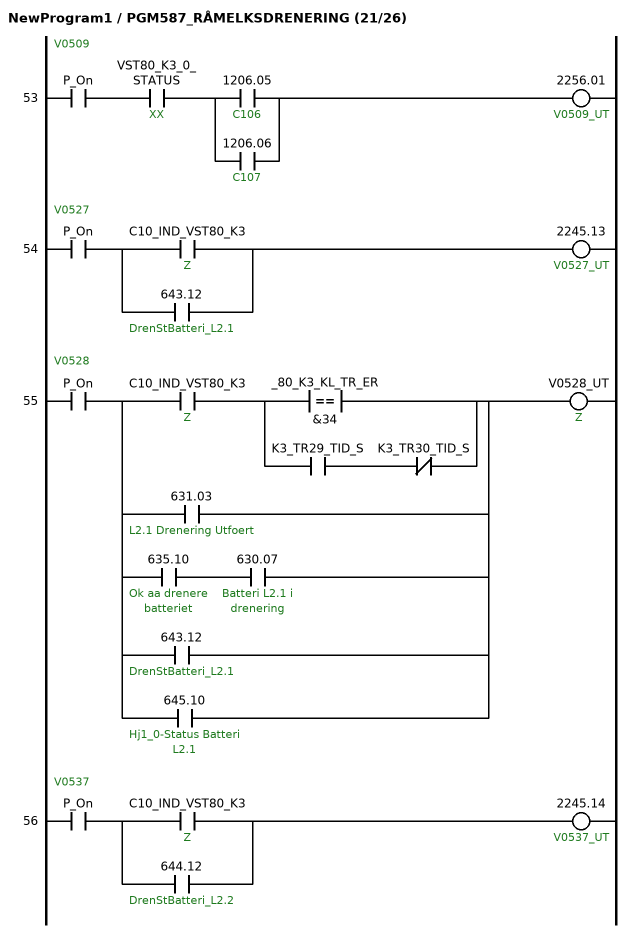
; rung 53: V0509
LD P_On
AND VST80_K3_0_STATUS  ; XX
LD 1206.05  ; C106
OR 1206.06  ; C107
ANDLD
OUT 2256.01  ; V0509_UT
; rung 54: V0527
LD P_On
LD C10_IND_VST80_K3  ; Z
OR 643.12  ; DrenStBatteri_L2.1
ANDLD
OUT 2245.13  ; V0527_UT
; rung 55: V0528
LD P_On
LD C10_IND_VST80_K3  ; Z
LD=(300) _80_K3_KL_TR_ER &34
LD K3_TR29_TID_S
ANDNOT K3_TR30_TID_S
ORLD
ANDLD
OR 631.03  ; L2.1 Drenering Utfoert
LD 635.10  ; Ok aa drenere batteriet
AND 630.07  ; Batteri L2.1 i drenering
ORLD
OR 643.12  ; DrenStBatteri_L2.1
OR 645.10  ; Hj1_0-Status Batteri L2.1
ANDLD
OUT V0528_UT  ; Z
; rung 56: V0537
LD P_On
LD C10_IND_VST80_K3  ; Z
OR 644.12  ; DrenStBatteri_L2.2
ANDLD
OUT 2245.14  ; V0537_UT

